// TIA Portal V17 export
// export: Created 2025-05-22T12:26:43.3929794Z, ExportSetting WithDefaults, DisplayName Totally Integrated Automation Portal, DisplayVersion V17 Update 8, DisplayName TIA Portal Openness, DisplayVersion V17 Update 8, DisplayName TIA Portal Version Control Interface, DisplayVersion V17, DisplayName SINAMICS Startdrive Advanced, DisplayVersion V17 SP2, DisplayName SINAMICS Startdrive G110M, G120, G120C, G120D, G120P, G115D, DisplayVersion V17 SP2, DisplayName SINAMICS Startdrive G130, G150, S120, S150, SINAMICS MV, S210, DisplayVersion V17 SP2, DisplayName STEP 7 Professional, DisplayVersion V17 Update 8, DisplayName SINUMERIK ONE STEP 7 Toolbox, DisplayVersion V17 Update 12, DisplayName SINUMERIK ONE PLC Basic Program Plus, DisplayVersion V17 Update 12, DisplayName SINUMERIK 840D sl STEP 7 Toolbox, DisplayVersion V17 Update 12, DisplayName STEP 7 Safety, DisplayVersion V17 Update 6, DisplayName WinCC Advanced, DisplayVersion V17 Update 8
FUNCTION "FC7453_QUALITY_PART_TYPE_CHANGE_CLADDING" : Void   // FC7453, LAD
{ S7_Optimized_Access := 'FALSE' }
AUTHOR : ETXETAR
NAME : GM-QC
VERSION : 1.0
// stored: AutoNumber false, IsIECCheckEnabled false, SetENOAutomatically false, UDAEnableTagReadback false
   VAR CONSTANT
      FC_NUMBER : DInt := 7453;
   END_VAR
   VAR_TEMP   // added for the SCL form of the ladder/FBD networks
      _w1 : Bool;
      _w2 : Bool;
   END_VAR
BEGIN

REGION Network 1: PART TYPE CHANGED AUXILIARY SET
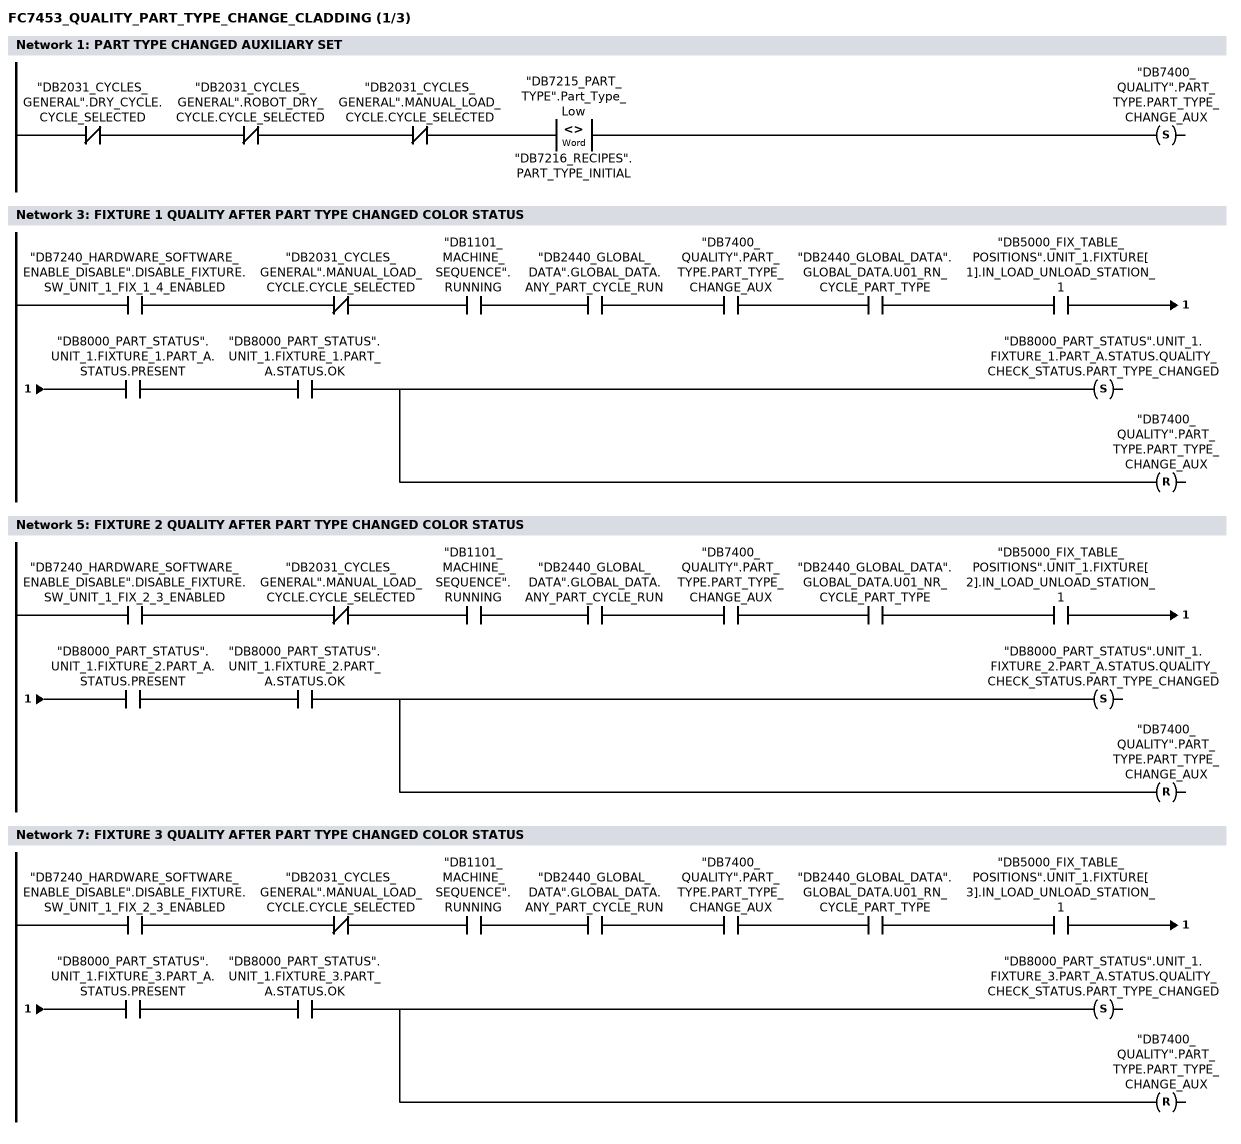
   RUNG wire#powerrail
      I_Contact( "DB2031_CYCLES_GENERAL".DRY_CYCLE.CYCLE_SELECTED )
      I_Contact( "DB2031_CYCLES_GENERAL".ROBOT_DRY_CYCLE.CYCLE_SELECTED )
      I_Contact( "DB2031_CYCLES_GENERAL".MANUAL_LOAD_CYCLE.CYCLE_SELECTED )
      { S7_Templates := "SrcType := Word" } NE_Contact(in1 := "DB7215_PART_TYPE".Part_Type_Low, in2 := "DB7216_RECIPES".PART_TYPE_INITIAL)
      S_Coil( "DB7400_QUALITY".PART_TYPE.PART_TYPE_CHANGE_AUX )
   END_RUNG
   // the same network as SCL:
   IF NOT "DB2031_CYCLES_GENERAL".DRY_CYCLE.CYCLE_SELECTED AND NOT "DB2031_CYCLES_GENERAL".ROBOT_DRY_CYCLE.CYCLE_SELECTED AND NOT "DB2031_CYCLES_GENERAL".MANUAL_LOAD_CYCLE.CYCLE_SELECTED AND ("DB7215_PART_TYPE".Part_Type_Low <> "DB7216_RECIPES".PART_TYPE_INITIAL) THEN
       "DB7400_QUALITY".PART_TYPE.PART_TYPE_CHANGE_AUX := TRUE;
   END_IF;
END_REGION

REGION Network 2: /////_FIXTURE_1_/////
END_REGION

REGION Network 3: FIXTURE 1 QUALITY AFTER PART TYPE CHANGED COLOR STATUS
   RUNG wire#powerrail
      Contact( "DB7240_HARDWARE_SOFTWARE_ENABLE_DISABLE".DISABLE_FIXTURE.SW_UNIT_1_FIX_1_4_ENABLED )
      I_Contact( "DB2031_CYCLES_GENERAL".MANUAL_LOAD_CYCLE.CYCLE_SELECTED )
      Contact( "DB1101_MACHINE_SEQUENCE".RUNNING )
      Contact( "DB2440_GLOBAL_DATA".GLOBAL_DATA.ANY_PART_CYCLE_RUN )
      Contact( "DB7400_QUALITY".PART_TYPE.PART_TYPE_CHANGE_AUX )
      Contact( "DB2440_GLOBAL_DATA".GLOBAL_DATA.U01_RN_CYCLE_PART_TYPE )
      Contact( "DB5000_FIX_TABLE_POSITIONS".UNIT_1.FIXTURE[1].IN_LOAD_UNLOAD_STATION_1 )
      Contact( "DB8000_PART_STATUS".UNIT_1.FIXTURE_1.PART_A.STATUS.PRESENT )
      Contact( "DB8000_PART_STATUS".UNIT_1.FIXTURE_1.PART_A.STATUS.OK )
      wire#w1
      S_Coil( "DB8000_PART_STATUS".UNIT_1.FIXTURE_1.PART_A.STATUS.QUALITY_CHECK_STATUS.PART_TYPE_CHANGED )
   END_RUNG
   RUNG wire#w1
      R_Coil( "DB7400_QUALITY".PART_TYPE.PART_TYPE_CHANGE_AUX )
   END_RUNG
   // the same network as SCL:
   IF "DB7240_HARDWARE_SOFTWARE_ENABLE_DISABLE".DISABLE_FIXTURE.SW_UNIT_1_FIX_1_4_ENABLED AND NOT "DB2031_CYCLES_GENERAL".MANUAL_LOAD_CYCLE.CYCLE_SELECTED AND "DB1101_MACHINE_SEQUENCE".RUNNING AND "DB2440_GLOBAL_DATA".GLOBAL_DATA.ANY_PART_CYCLE_RUN AND "DB7400_QUALITY".PART_TYPE.PART_TYPE_CHANGE_AUX AND "DB2440_GLOBAL_DATA".GLOBAL_DATA.U01_RN_CYCLE_PART_TYPE AND "DB5000_FIX_TABLE_POSITIONS".UNIT_1.FIXTURE[1].IN_LOAD_UNLOAD_STATION_1 AND "DB8000_PART_STATUS".UNIT_1.FIXTURE_1.PART_A.STATUS.PRESENT AND "DB8000_PART_STATUS".UNIT_1.FIXTURE_1.PART_A.STATUS.OK THEN
       "DB8000_PART_STATUS".UNIT_1.FIXTURE_1.PART_A.STATUS.QUALITY_CHECK_STATUS.PART_TYPE_CHANGED := TRUE;
       "DB7400_QUALITY".PART_TYPE.PART_TYPE_CHANGE_AUX := FALSE;
   END_IF;
END_REGION

REGION Network 4: /////_FIXTURE_2_/////
END_REGION

REGION Network 5: FIXTURE 2 QUALITY AFTER PART TYPE CHANGED COLOR STATUS
   RUNG wire#powerrail
      Contact( "DB7240_HARDWARE_SOFTWARE_ENABLE_DISABLE".DISABLE_FIXTURE.SW_UNIT_1_FIX_2_3_ENABLED )
      I_Contact( "DB2031_CYCLES_GENERAL".MANUAL_LOAD_CYCLE.CYCLE_SELECTED )
      Contact( "DB1101_MACHINE_SEQUENCE".RUNNING )
      Contact( "DB2440_GLOBAL_DATA".GLOBAL_DATA.ANY_PART_CYCLE_RUN )
      Contact( "DB7400_QUALITY".PART_TYPE.PART_TYPE_CHANGE_AUX )
      Contact( "DB2440_GLOBAL_DATA".GLOBAL_DATA.U01_NR_CYCLE_PART_TYPE )
      Contact( "DB5000_FIX_TABLE_POSITIONS".UNIT_1.FIXTURE[2].IN_LOAD_UNLOAD_STATION_1 )
      Contact( "DB8000_PART_STATUS".UNIT_1.FIXTURE_2.PART_A.STATUS.PRESENT )
      Contact( "DB8000_PART_STATUS".UNIT_1.FIXTURE_2.PART_A.STATUS.OK )
      wire#w1
      S_Coil( "DB8000_PART_STATUS".UNIT_1.FIXTURE_2.PART_A.STATUS.QUALITY_CHECK_STATUS.PART_TYPE_CHANGED )
   END_RUNG
   RUNG wire#w1
      R_Coil( "DB7400_QUALITY".PART_TYPE.PART_TYPE_CHANGE_AUX )
   END_RUNG
   // the same network as SCL:
   IF "DB7240_HARDWARE_SOFTWARE_ENABLE_DISABLE".DISABLE_FIXTURE.SW_UNIT_1_FIX_2_3_ENABLED AND NOT "DB2031_CYCLES_GENERAL".MANUAL_LOAD_CYCLE.CYCLE_SELECTED AND "DB1101_MACHINE_SEQUENCE".RUNNING AND "DB2440_GLOBAL_DATA".GLOBAL_DATA.ANY_PART_CYCLE_RUN AND "DB7400_QUALITY".PART_TYPE.PART_TYPE_CHANGE_AUX AND "DB2440_GLOBAL_DATA".GLOBAL_DATA.U01_NR_CYCLE_PART_TYPE AND "DB5000_FIX_TABLE_POSITIONS".UNIT_1.FIXTURE[2].IN_LOAD_UNLOAD_STATION_1 AND "DB8000_PART_STATUS".UNIT_1.FIXTURE_2.PART_A.STATUS.PRESENT AND "DB8000_PART_STATUS".UNIT_1.FIXTURE_2.PART_A.STATUS.OK THEN
       "DB8000_PART_STATUS".UNIT_1.FIXTURE_2.PART_A.STATUS.QUALITY_CHECK_STATUS.PART_TYPE_CHANGED := TRUE;
       "DB7400_QUALITY".PART_TYPE.PART_TYPE_CHANGE_AUX := FALSE;
   END_IF;
END_REGION

REGION Network 6: /////_FIXTURE_3_/////
END_REGION

REGION Network 7: FIXTURE 3 QUALITY AFTER PART TYPE CHANGED COLOR STATUS
   RUNG wire#powerrail
      Contact( "DB7240_HARDWARE_SOFTWARE_ENABLE_DISABLE".DISABLE_FIXTURE.SW_UNIT_1_FIX_2_3_ENABLED )
      I_Contact( "DB2031_CYCLES_GENERAL".MANUAL_LOAD_CYCLE.CYCLE_SELECTED )
      Contact( "DB1101_MACHINE_SEQUENCE".RUNNING )
      Contact( "DB2440_GLOBAL_DATA".GLOBAL_DATA.ANY_PART_CYCLE_RUN )
      Contact( "DB7400_QUALITY".PART_TYPE.PART_TYPE_CHANGE_AUX )
      Contact( "DB2440_GLOBAL_DATA".GLOBAL_DATA.U01_RN_CYCLE_PART_TYPE )
      Contact( "DB5000_FIX_TABLE_POSITIONS".UNIT_1.FIXTURE[3].IN_LOAD_UNLOAD_STATION_1 )
      Contact( "DB8000_PART_STATUS".UNIT_1.FIXTURE_3.PART_A.STATUS.PRESENT )
      Contact( "DB8000_PART_STATUS".UNIT_1.FIXTURE_3.PART_A.STATUS.OK )
      wire#w1
      S_Coil( "DB8000_PART_STATUS".UNIT_1.FIXTURE_3.PART_A.STATUS.QUALITY_CHECK_STATUS.PART_TYPE_CHANGED )
   END_RUNG
   RUNG wire#w1
      R_Coil( "DB7400_QUALITY".PART_TYPE.PART_TYPE_CHANGE_AUX )
   END_RUNG
   // the same network as SCL:
   IF "DB7240_HARDWARE_SOFTWARE_ENABLE_DISABLE".DISABLE_FIXTURE.SW_UNIT_1_FIX_2_3_ENABLED AND NOT "DB2031_CYCLES_GENERAL".MANUAL_LOAD_CYCLE.CYCLE_SELECTED AND "DB1101_MACHINE_SEQUENCE".RUNNING AND "DB2440_GLOBAL_DATA".GLOBAL_DATA.ANY_PART_CYCLE_RUN AND "DB7400_QUALITY".PART_TYPE.PART_TYPE_CHANGE_AUX AND "DB2440_GLOBAL_DATA".GLOBAL_DATA.U01_RN_CYCLE_PART_TYPE AND "DB5000_FIX_TABLE_POSITIONS".UNIT_1.FIXTURE[3].IN_LOAD_UNLOAD_STATION_1 AND "DB8000_PART_STATUS".UNIT_1.FIXTURE_3.PART_A.STATUS.PRESENT AND "DB8000_PART_STATUS".UNIT_1.FIXTURE_3.PART_A.STATUS.OK THEN
       "DB8000_PART_STATUS".UNIT_1.FIXTURE_3.PART_A.STATUS.QUALITY_CHECK_STATUS.PART_TYPE_CHANGED := TRUE;
       "DB7400_QUALITY".PART_TYPE.PART_TYPE_CHANGE_AUX := FALSE;
   END_IF;
END_REGION

REGION Network 8: /////_FIXTURE_4_/////
END_REGION

REGION Network 9: FIXTURE 4 QUALITY AFTER PART TYPE CHANGED COLOR STATUS
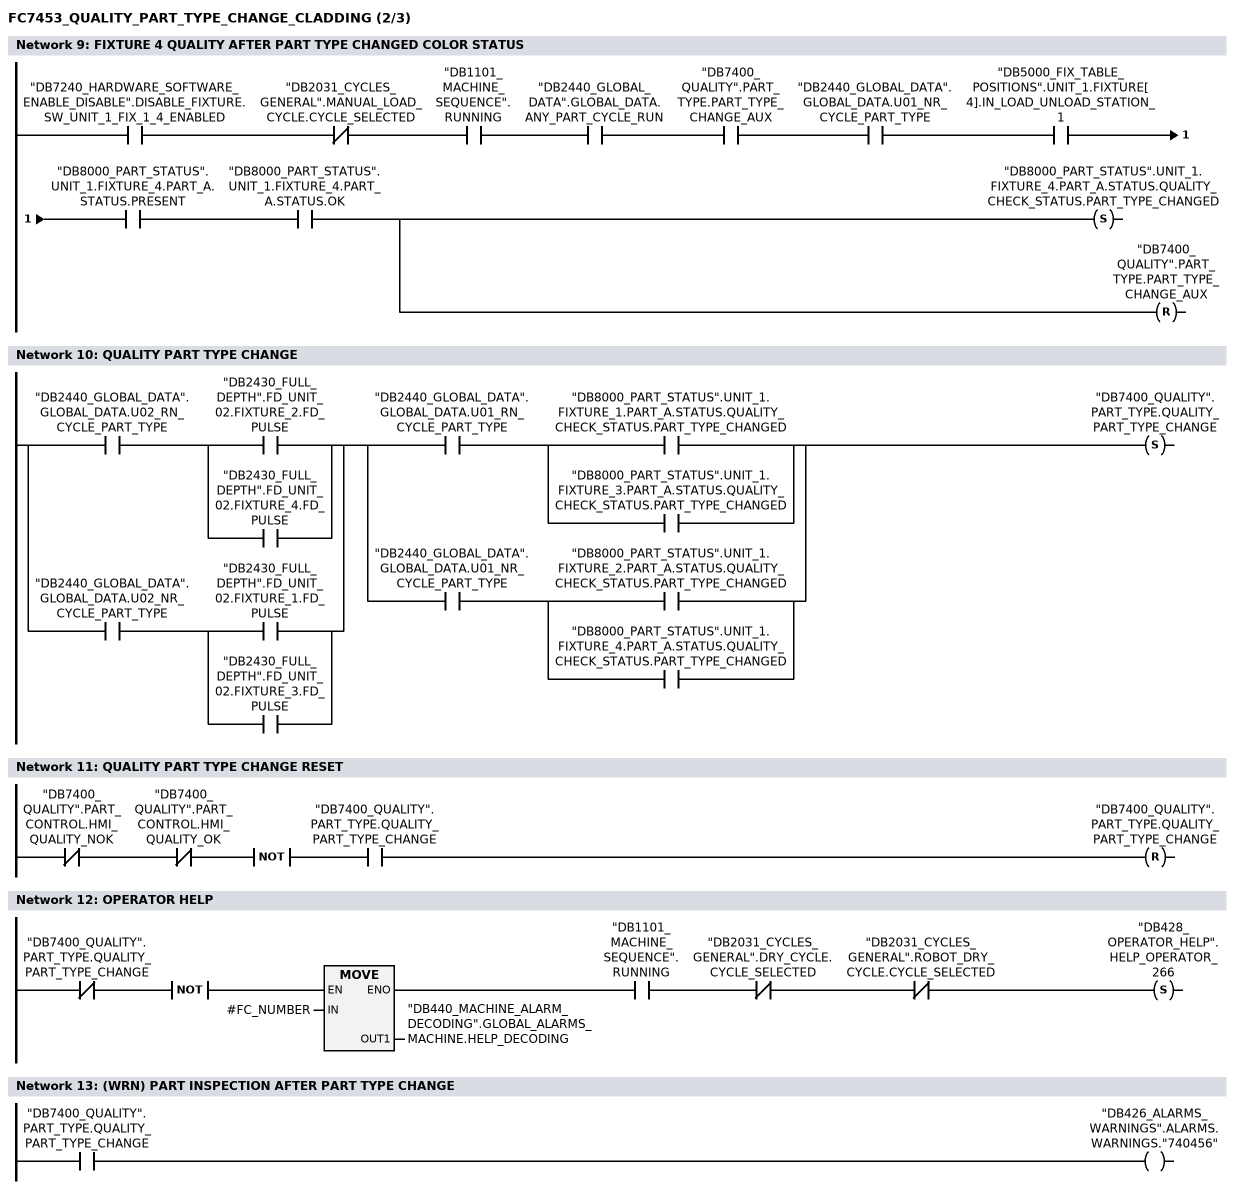
   RUNG wire#powerrail
      Contact( "DB7240_HARDWARE_SOFTWARE_ENABLE_DISABLE".DISABLE_FIXTURE.SW_UNIT_1_FIX_1_4_ENABLED )
      I_Contact( "DB2031_CYCLES_GENERAL".MANUAL_LOAD_CYCLE.CYCLE_SELECTED )
      Contact( "DB1101_MACHINE_SEQUENCE".RUNNING )
      Contact( "DB2440_GLOBAL_DATA".GLOBAL_DATA.ANY_PART_CYCLE_RUN )
      Contact( "DB7400_QUALITY".PART_TYPE.PART_TYPE_CHANGE_AUX )
      Contact( "DB2440_GLOBAL_DATA".GLOBAL_DATA.U01_NR_CYCLE_PART_TYPE )
      Contact( "DB5000_FIX_TABLE_POSITIONS".UNIT_1.FIXTURE[4].IN_LOAD_UNLOAD_STATION_1 )
      Contact( "DB8000_PART_STATUS".UNIT_1.FIXTURE_4.PART_A.STATUS.PRESENT )
      Contact( "DB8000_PART_STATUS".UNIT_1.FIXTURE_4.PART_A.STATUS.OK )
      wire#w1
      S_Coil( "DB8000_PART_STATUS".UNIT_1.FIXTURE_4.PART_A.STATUS.QUALITY_CHECK_STATUS.PART_TYPE_CHANGED )
   END_RUNG
   RUNG wire#w1
      R_Coil( "DB7400_QUALITY".PART_TYPE.PART_TYPE_CHANGE_AUX )
   END_RUNG
   // the same network as SCL:
   IF "DB7240_HARDWARE_SOFTWARE_ENABLE_DISABLE".DISABLE_FIXTURE.SW_UNIT_1_FIX_1_4_ENABLED AND NOT "DB2031_CYCLES_GENERAL".MANUAL_LOAD_CYCLE.CYCLE_SELECTED AND "DB1101_MACHINE_SEQUENCE".RUNNING AND "DB2440_GLOBAL_DATA".GLOBAL_DATA.ANY_PART_CYCLE_RUN AND "DB7400_QUALITY".PART_TYPE.PART_TYPE_CHANGE_AUX AND "DB2440_GLOBAL_DATA".GLOBAL_DATA.U01_NR_CYCLE_PART_TYPE AND "DB5000_FIX_TABLE_POSITIONS".UNIT_1.FIXTURE[4].IN_LOAD_UNLOAD_STATION_1 AND "DB8000_PART_STATUS".UNIT_1.FIXTURE_4.PART_A.STATUS.PRESENT AND "DB8000_PART_STATUS".UNIT_1.FIXTURE_4.PART_A.STATUS.OK THEN
       "DB8000_PART_STATUS".UNIT_1.FIXTURE_4.PART_A.STATUS.QUALITY_CHECK_STATUS.PART_TYPE_CHANGED := TRUE;
       "DB7400_QUALITY".PART_TYPE.PART_TYPE_CHANGE_AUX := FALSE;
   END_IF;
END_REGION

REGION Network 10: QUALITY PART TYPE CHANGE
   RUNG wire#powerrail
      Contact( "DB2440_GLOBAL_DATA".GLOBAL_DATA.U02_RN_CYCLE_PART_TYPE )
      wire#w1
      Contact( "DB2430_FULL_DEPTH".FD_UNIT_02.FIXTURE_2.FD_PULSE )
      wire#w2
      Contact( "DB2440_GLOBAL_DATA".GLOBAL_DATA.U01_RN_CYCLE_PART_TYPE )
      wire#w4
      Contact( "DB8000_PART_STATUS".UNIT_1.FIXTURE_1.PART_A.STATUS.QUALITY_CHECK_STATUS.PART_TYPE_CHANGED )
      wire#w5
      S_Coil( "DB7400_QUALITY".PART_TYPE.QUALITY_PART_TYPE_CHANGE )
   END_RUNG
   RUNG wire#w1
      Contact( "DB2430_FULL_DEPTH".FD_UNIT_02.FIXTURE_4.FD_PULSE )
   END_RUNG wire#w2
   RUNG wire#powerrail
      Contact( "DB2440_GLOBAL_DATA".GLOBAL_DATA.U02_NR_CYCLE_PART_TYPE )
      wire#w3
      Contact( "DB2430_FULL_DEPTH".FD_UNIT_02.FIXTURE_1.FD_PULSE )
   END_RUNG wire#w2
   RUNG wire#w3
      Contact( "DB2430_FULL_DEPTH".FD_UNIT_02.FIXTURE_3.FD_PULSE )
   END_RUNG wire#w2
   RUNG wire#w4
      Contact( "DB8000_PART_STATUS".UNIT_1.FIXTURE_3.PART_A.STATUS.QUALITY_CHECK_STATUS.PART_TYPE_CHANGED )
   END_RUNG wire#w5
   RUNG wire#w2
      Contact( "DB2440_GLOBAL_DATA".GLOBAL_DATA.U01_NR_CYCLE_PART_TYPE )
      wire#w6
      Contact( "DB8000_PART_STATUS".UNIT_1.FIXTURE_2.PART_A.STATUS.QUALITY_CHECK_STATUS.PART_TYPE_CHANGED )
   END_RUNG wire#w5
   RUNG wire#w6
      Contact( "DB8000_PART_STATUS".UNIT_1.FIXTURE_4.PART_A.STATUS.QUALITY_CHECK_STATUS.PART_TYPE_CHANGED )
   END_RUNG wire#w5
   // the same network as SCL:
   IF (("DB2440_GLOBAL_DATA".GLOBAL_DATA.U02_RN_CYCLE_PART_TYPE AND ("DB2430_FULL_DEPTH".FD_UNIT_02.FIXTURE_2.FD_PULSE OR "DB2430_FULL_DEPTH".FD_UNIT_02.FIXTURE_4.FD_PULSE)) OR ("DB2440_GLOBAL_DATA".GLOBAL_DATA.U02_NR_CYCLE_PART_TYPE AND ("DB2430_FULL_DEPTH".FD_UNIT_02.FIXTURE_1.FD_PULSE OR "DB2430_FULL_DEPTH".FD_UNIT_02.FIXTURE_3.FD_PULSE))) AND (("DB2440_GLOBAL_DATA".GLOBAL_DATA.U01_RN_CYCLE_PART_TYPE AND ("DB8000_PART_STATUS".UNIT_1.FIXTURE_1.PART_A.STATUS.QUALITY_CHECK_STATUS.PART_TYPE_CHANGED OR "DB8000_PART_STATUS".UNIT_1.FIXTURE_3.PART_A.STATUS.QUALITY_CHECK_STATUS.PART_TYPE_CHANGED)) OR ("DB2440_GLOBAL_DATA".GLOBAL_DATA.U01_NR_CYCLE_PART_TYPE AND ("DB8000_PART_STATUS".UNIT_1.FIXTURE_2.PART_A.STATUS.QUALITY_CHECK_STATUS.PART_TYPE_CHANGED OR "DB8000_PART_STATUS".UNIT_1.FIXTURE_4.PART_A.STATUS.QUALITY_CHECK_STATUS.PART_TYPE_CHANGED))) THEN
       "DB7400_QUALITY".PART_TYPE.QUALITY_PART_TYPE_CHANGE := TRUE;
   END_IF;
END_REGION

REGION Network 11: QUALITY PART TYPE CHANGE RESET
   RUNG wire#powerrail
      I_Contact( "DB7400_QUALITY".PART_CONTROL.HMI_QUALITY_NOK )
      I_Contact( "DB7400_QUALITY".PART_CONTROL.HMI_QUALITY_OK )
      Not()
      Contact( "DB7400_QUALITY".PART_TYPE.QUALITY_PART_TYPE_CHANGE )
      R_Coil( "DB7400_QUALITY".PART_TYPE.QUALITY_PART_TYPE_CHANGE )
   END_RUNG
   // the same network as SCL:
   IF NOT (NOT "DB7400_QUALITY".PART_CONTROL.HMI_QUALITY_NOK AND NOT "DB7400_QUALITY".PART_CONTROL.HMI_QUALITY_OK) AND "DB7400_QUALITY".PART_TYPE.QUALITY_PART_TYPE_CHANGE THEN
       "DB7400_QUALITY".PART_TYPE.QUALITY_PART_TYPE_CHANGE := FALSE;
   END_IF;
END_REGION

REGION Network 12: OPERATOR HELP
   RUNG wire#powerrail
      I_Contact( "DB7400_QUALITY".PART_TYPE.QUALITY_PART_TYPE_CHANGE )
      Not()
      { S7_GenerateENO := "TRUE" } Move(in := #FC_NUMBER, out1 => "DB440_MACHINE_ALARM_DECODING".GLOBAL_ALARMS_MACHINE.HELP_DECODING)
      Contact( "DB1101_MACHINE_SEQUENCE".RUNNING )
      I_Contact( "DB2031_CYCLES_GENERAL".DRY_CYCLE.CYCLE_SELECTED )
      I_Contact( "DB2031_CYCLES_GENERAL".ROBOT_DRY_CYCLE.CYCLE_SELECTED )
      S_Coil( "DB428_OPERATOR_HELP".HELP_OPERATOR_266 )
   END_RUNG
   // the same network as SCL:
   // ENO of a box is taken as its EN; it also drops when the box reports an error
   #_w1 := NOT (NOT "DB7400_QUALITY".PART_TYPE.QUALITY_PART_TYPE_CHANGE);
   IF #_w1 THEN "DB440_MACHINE_ALARM_DECODING".GLOBAL_ALARMS_MACHINE.HELP_DECODING := #FC_NUMBER; END_IF;
   IF #_w1 AND "DB1101_MACHINE_SEQUENCE".RUNNING AND NOT "DB2031_CYCLES_GENERAL".DRY_CYCLE.CYCLE_SELECTED AND NOT "DB2031_CYCLES_GENERAL".ROBOT_DRY_CYCLE.CYCLE_SELECTED THEN
       "DB428_OPERATOR_HELP".HELP_OPERATOR_266 := TRUE;
   END_IF;
END_REGION

REGION Network 13: (WRN) PART INSPECTION AFTER PART TYPE CHANGE
   RUNG wire#powerrail
      Contact( "DB7400_QUALITY".PART_TYPE.QUALITY_PART_TYPE_CHANGE )
      Coil( "DB426_ALARMS_WARNINGS".ALARMS.WARNINGS."740456" )
   END_RUNG
   // the same network as SCL:
   "DB426_ALARMS_WARNINGS".ALARMS.WARNINGS."740456" := "DB7400_QUALITY".PART_TYPE.QUALITY_PART_TYPE_CHANGE;
END_REGION

REGION Network 14: QUALITY AFTER PART TYPE CHANGE NOK ALARM
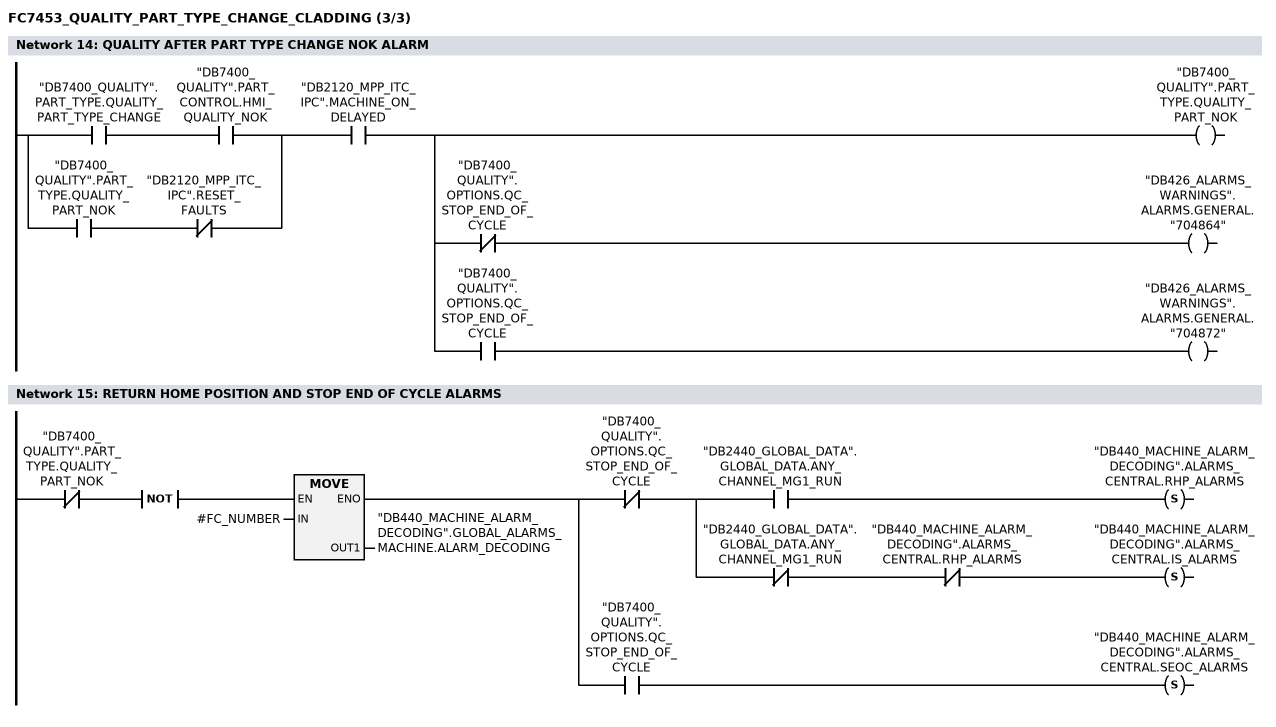
   RUNG wire#powerrail
      Contact( "DB7400_QUALITY".PART_TYPE.QUALITY_PART_TYPE_CHANGE )
      Contact( "DB7400_QUALITY".PART_CONTROL.HMI_QUALITY_NOK )
      wire#w1
      Contact( "DB2120_MPP_ITC_IPC".MACHINE_ON_DELAYED )
      wire#w2
      Coil( "DB7400_QUALITY".PART_TYPE.QUALITY_PART_NOK )
   END_RUNG
   RUNG wire#powerrail
      Contact( "DB7400_QUALITY".PART_TYPE.QUALITY_PART_NOK )
      I_Contact( "DB2120_MPP_ITC_IPC".RESET_FAULTS )
   END_RUNG wire#w1
   RUNG wire#w2
      I_Contact( "DB7400_QUALITY".OPTIONS.QC_STOP_END_OF_CYCLE )
      Coil( "DB426_ALARMS_WARNINGS".ALARMS.GENERAL."704864" )
   END_RUNG
   RUNG wire#w2
      Contact( "DB7400_QUALITY".OPTIONS.QC_STOP_END_OF_CYCLE )
      Coil( "DB426_ALARMS_WARNINGS".ALARMS.GENERAL."704872" )
   END_RUNG
   // the same network as SCL:
   "DB7400_QUALITY".PART_TYPE.QUALITY_PART_NOK := (("DB7400_QUALITY".PART_TYPE.QUALITY_PART_TYPE_CHANGE AND "DB7400_QUALITY".PART_CONTROL.HMI_QUALITY_NOK) OR ("DB7400_QUALITY".PART_TYPE.QUALITY_PART_NOK AND NOT "DB2120_MPP_ITC_IPC".RESET_FAULTS)) AND "DB2120_MPP_ITC_IPC".MACHINE_ON_DELAYED;
   "DB426_ALARMS_WARNINGS".ALARMS.GENERAL."704864" := "DB7400_QUALITY".PART_TYPE.QUALITY_PART_NOK AND NOT "DB7400_QUALITY".OPTIONS.QC_STOP_END_OF_CYCLE;
   "DB426_ALARMS_WARNINGS".ALARMS.GENERAL."704872" := "DB7400_QUALITY".PART_TYPE.QUALITY_PART_NOK AND "DB7400_QUALITY".OPTIONS.QC_STOP_END_OF_CYCLE;
END_REGION

REGION Network 15: RETURN HOME POSITION AND STOP END OF CYCLE ALARMS
   RUNG wire#powerrail
      I_Contact( "DB7400_QUALITY".PART_TYPE.QUALITY_PART_NOK )
      Not()
      { S7_GenerateENO := "TRUE" } Move(in := #FC_NUMBER, out1 => "DB440_MACHINE_ALARM_DECODING".GLOBAL_ALARMS_MACHINE.ALARM_DECODING)
      wire#w1
      I_Contact( "DB7400_QUALITY".OPTIONS.QC_STOP_END_OF_CYCLE )
      wire#w2
      Contact( "DB2440_GLOBAL_DATA".GLOBAL_DATA.ANY_CHANNEL_MG1_RUN )
      S_Coil( "DB440_MACHINE_ALARM_DECODING".ALARMS_CENTRAL.RHP_ALARMS )
   END_RUNG
   RUNG wire#w2
      I_Contact( "DB2440_GLOBAL_DATA".GLOBAL_DATA.ANY_CHANNEL_MG1_RUN )
      I_Contact( "DB440_MACHINE_ALARM_DECODING".ALARMS_CENTRAL.RHP_ALARMS )
      S_Coil( "DB440_MACHINE_ALARM_DECODING".ALARMS_CENTRAL.IS_ALARMS )
   END_RUNG
   RUNG wire#w1
      Contact( "DB7400_QUALITY".OPTIONS.QC_STOP_END_OF_CYCLE )
      S_Coil( "DB440_MACHINE_ALARM_DECODING".ALARMS_CENTRAL.SEOC_ALARMS )
   END_RUNG
   // the same network as SCL:
   // ENO of a box is taken as its EN; it also drops when the box reports an error
   #_w1 := NOT (NOT "DB7400_QUALITY".PART_TYPE.QUALITY_PART_NOK);
   IF #_w1 THEN "DB440_MACHINE_ALARM_DECODING".GLOBAL_ALARMS_MACHINE.ALARM_DECODING := #FC_NUMBER; END_IF;
   #_w2 := #_w1 AND NOT "DB7400_QUALITY".OPTIONS.QC_STOP_END_OF_CYCLE;
   IF #_w2 AND "DB2440_GLOBAL_DATA".GLOBAL_DATA.ANY_CHANNEL_MG1_RUN THEN
       "DB440_MACHINE_ALARM_DECODING".ALARMS_CENTRAL.RHP_ALARMS := TRUE;
   END_IF;
   IF #_w2 AND NOT "DB2440_GLOBAL_DATA".GLOBAL_DATA.ANY_CHANNEL_MG1_RUN AND NOT "DB440_MACHINE_ALARM_DECODING".ALARMS_CENTRAL.RHP_ALARMS THEN
       "DB440_MACHINE_ALARM_DECODING".ALARMS_CENTRAL.IS_ALARMS := TRUE;
   END_IF;
   IF #_w1 AND "DB7400_QUALITY".OPTIONS.QC_STOP_END_OF_CYCLE THEN
       "DB440_MACHINE_ALARM_DECODING".ALARMS_CENTRAL.SEOC_ALARMS := TRUE;
   END_IF;
END_REGION
END_FUNCTION
